KUKA KRL program: safety_test_01.src, safety_test_01.dat

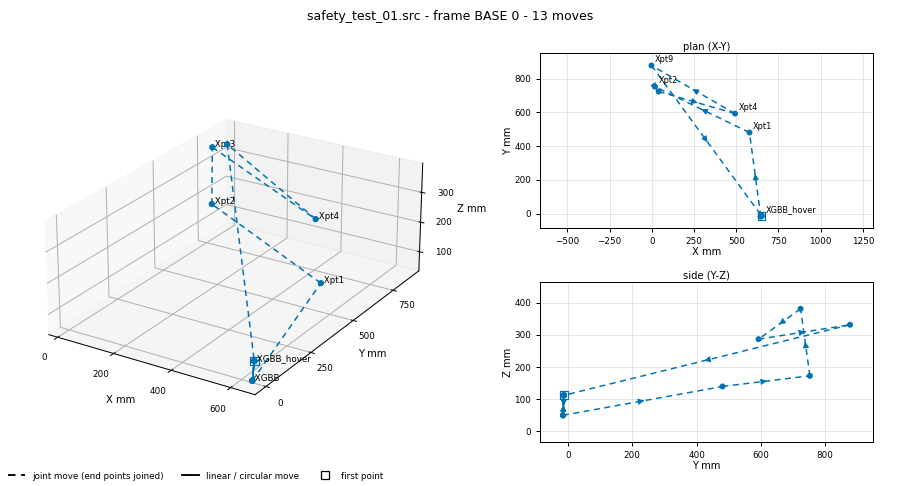
[picture p0: tool path of safety_test_01.src in frame BASE 0, 13 of 13 moves have a stored position in this frame; points joined in program order, loops and branches not executed]
--- safety_test_01.src ---
&ACCESS RVP
&REL 80
&PARAM TEMPLATE = C:\KRC\Roboter\Template\vorgabe
&PARAM EDITMASK = *
DEF safety_test_01( )

DECL INT COUNT
DECL INT MODE
DECL INT POSITION
DECL BOOL PREEMPT
DECL BOOL SICK_TEST
DECL BOOL STOP_TEST
DECL BOOL MOVING

;FOLD INI
  ;FOLD BASISTECH INI
    GLOBAL INTERRUPT DECL 3 WHEN $STOPMESS==TRUE DO IR_STOPM ( )
    INTERRUPT ON 3
    BAS (#INITMOV,0 )
  ;ENDFOLD (BASISTECH INI)
  ;FOLD USER INI
    ;Make your modifications here

  ;ENDFOLD (USER INI)
;ENDFOLD (INI)

; Start motions at the hover point
;FOLD PTP GBB_hover Vel=100 % PDAT1 Tool[4]:Pneumatic_gripper Base[0];%{PE}%R 5.6.11,%MKUKATPBASIS,%CMOVE,%VPTP,%P 1:PTP, 2:GBB_hover, 3:, 5:100, 7:PDAT1
$BWDSTART=FALSE
PDAT_ACT=PPDAT1
FDAT_ACT=FGBB_hover
BAS(#PTP_PARAMS,100)
PTP XGBB_hover
;ENDFOLD

MOVING=true
MODE = 4
POSITION = 1
PREEMPT = true
SICK_TEST = FALSE
STOP_TEST = FALSE

SWITCH MODE
  CASE 0
   ; SToP TeSt
   STOP_TEST = TRUE

  CASE 1
    ; Safety rated monitored stop
    OVERRIDE_SPEED = TRUE
    MOVE_PERMISSION = FALSE
  CASE 2
    ; Give permission for robot to move
    MOVE_PERMISSION = TRUE
    OVERRIDE_SPEED = FALSE
  CASE 3
    ; test 1
    MOVE_PERMISSION = FALSE
    OVERRIDE_SPEED = FALSe
  CASE 4
    ; full test
    OVERRIDE_SPEED = TRUE
    MOVE_PERMISSION = true
ENDSWITCH



; Move to button
;FOLD LIN GBB Vel=0.5 m/s CPDAT4 Tool[4]:Pneumatic_gripper Base[0];%{PE}%R 5.6.11,%MKUKATPBASIS,%CMOVE,%VLIN,%P 1:LIN, 2:GBB, 3:, 5:0.5, 7:CPDAT4
$BWDSTART=FALSE
LDAT_ACT=LCPDAT4
FDAT_ACT=FGBB
BAS(#CP_PARAMS,0.5)
LIN XGBB
;ENDFOLD

HALT

;FOLD WAIT Time=15 sec;%{PE}%R 5.6.11,%MKUKATPBASIS,%CWAIT,%VWAIT,%P 2:15
WAIT SEC 15
;ENDFOLD

; 2 stow request
; 3 robot can move
; 4 agv stopped
; 5 agv stopped verify
; 6 sick signal

IF SICK_TEST THEN
  WHILE TRUE
    IF $IN[6] THEN
      $OUT[1] = FALSE
    ELSE
      $OUT[1] = TRUE
    ENDIF
  ENDWHILE
ELSE
  IF MOVE_PERMISSION OR STOP_TEST THEN
;    $OUT[1] = TRUE
    IF MOVE_PERMISSION THEN
      ; Permission to move
      WAIT FOR ($IN[3])
    ENDIF
    ; Verification is safe to move
    WAIT FOR ($IN[4] and not $IN[5])

;    WAIT FOR ($IN[4])
  ENDIF

  ;FOLD PTP GBB_hover Vel=100 % PDAT15 Tool[4]:Pneumatic_gripper Base[0];%{PE}%R 5.6.11,%MKUKATPBASIS,%CMOVE,%VPTP,%P 1:PTP, 2:GBB_hover, 3:, 5:100, 7:PDAT15
$BWDSTART=FALSE
PDAT_ACT=PPDAT15
FDAT_ACT=FGBB_hover
BAS(#PTP_PARAMS,100)
PTP XGBB_hover
;ENDFOLD

;  HALT

  FOR COUNT = 1 TO 80
    ; Allow AGV to preempt motion
    IF (PREEMPT AND MOVE_PERMISSION) OR (STOP_TEST AND $IN[5]) THEN
      IF $IN[2] OR (STOP_TEST AND $IN[5]) THEN
;        PTP GBB_HOVER C_PTP

        ;FOLD PTP GBB_hover Vel=100 % PDAT16 Tool[4]:Pneumatic_gripper Base[0];%{PE}%R 5.6.11,%MKUKATPBASIS,%CMOVE,%VPTP,%P 1:PTP, 2:GBB_hover, 3:, 5:100, 7:PDAT16
$BWDSTART=FALSE
PDAT_ACT=PPDAT16
FDAT_ACT=FGBB_hover
BAS(#PTP_PARAMS,100)
PTP XGBB_hover
;ENDFOLD
;        LIN GBB

        ;FOLD LIN GBB Vel=0.5 m/s CPDAT5 Tool[4]:Pneumatic_gripper Base[0];%{PE}%R 5.6.11,%MKUKATPBASIS,%CMOVE,%VLIN,%P 1:LIN, 2:GBB, 3:, 5:0.5, 7:CPDAT5
$BWDSTART=FALSE
LDAT_ACT=LCPDAT5
FDAT_ACT=FGBB
BAS(#CP_PARAMS,0.5)
LIN XGBB
;ENDFOLD
        IF MOVE_PERMISSION THEN
          WAIT FOR ((NOT $IN[2]) and ($IN[3]))
        ELSE
          WAIT FOR ($IN[4] AND NOT $IN[5])
        ENDIF
      ENDIF
    ENDIF

    IF MOVING THEN
      SWITCH POSITION
      CASE 1
        ;FOLD PTP pt1 CONT Vel=50 % PDAT10 Tool[4]:Pneumatic_gripper Base[0];%{PE}%R 5.6.11,%MKUKATPBASIS,%CMOVE,%VPTP,%P 1:PTP, 2:pt1, 3:C_PTP, 5:50, 7:PDAT10
$BWDSTART=FALSE
PDAT_ACT=PPDAT10
FDAT_ACT=Fpt1
BAS(#PTP_PARAMS,50)
PTP Xpt1 C_PTP
;ENDFOLD
        POSITION = 2
      CASE 2
        ;FOLD PTP pt2 CONT Vel=50 % PDAT11 Tool[4]:Pneumatic_gripper Base[0];%{PE}%R 5.6.11,%MKUKATPBASIS,%CMOVE,%VPTP,%P 1:PTP, 2:pt2, 3:C_PTP, 5:50, 7:PDAT11
$BWDSTART=FALSE
PDAT_ACT=PPDAT11
FDAT_ACT=Fpt2
BAS(#PTP_PARAMS,50)
PTP Xpt2 C_PTP
;ENDFOLD
        POSITION = 3
      CASE 3
        ;FOLD PTP pt3 CONT Vel=50 % PDAT12 Tool[4]:Pneumatic_gripper Base[0];%{PE}%R 5.6.11,%MKUKATPBASIS,%CMOVE,%VPTP,%P 1:PTP, 2:pt3, 3:C_PTP, 5:50, 7:PDAT12
$BWDSTART=FALSE
PDAT_ACT=PPDAT12
FDAT_ACT=Fpt3
BAS(#PTP_PARAMS,50)
PTP Xpt3 C_PTP
;ENDFOLD
        POSITION = 4
      CASE 4
        ;FOLD PTP pt4 CONT Vel=50 % PDAT13 Tool[4]:Pneumatic_gripper Base[0];%{PE}%R 5.6.11,%MKUKATPBASIS,%CMOVE,%VPTP,%P 1:PTP, 2:pt4, 3:C_PTP, 5:50, 7:PDAT13
$BWDSTART=FALSE
PDAT_ACT=PPDAT13
FDAT_ACT=Fpt4
BAS(#PTP_PARAMS,50)
PTP Xpt4 C_PTP
;ENDFOLD
        POSITION = 1
      ENDSWITCH
    ELSE

;FOLD PTP pt9 Vel=50 % PDAT17 Tool[1]:flange_adapter Base[0];%{PE}%R 5.6.11,%MKUKATPBASIS,%CMOVE,%VPTP,%P 1:PTP, 2:pt9, 3:, 5:50, 7:PDAT17
$BWDSTART=FALSE
PDAT_ACT=PPDAT17
FDAT_ACT=Fpt9
BAS(#PTP_PARAMS,50)
PTP Xpt9
;ENDFOLD
    ENDIF
  ENDFOR


  $OUT[1] = FALSE
ENDIF

; move back to button
;FOLD PTP GBB_hover Vel=100 % PDAT9 Tool[4]:Pneumatic_gripper Base[0];%{PE}%R 5.6.11,%MKUKATPBASIS,%CMOVE,%VPTP,%P 1:PTP, 2:GBB_hover, 3:, 5:100, 7:PDAT9
$BWDSTART=FALSE
PDAT_ACT=PPDAT9
FDAT_ACT=FGBB_hover
BAS(#PTP_PARAMS,100)
PTP XGBB_hover
;ENDFOLD

;FOLD LIN GBB Vel=0.5 m/s CPDAT1 Tool[4]:Pneumatic_gripper Base[0];%{PE}%R 5.6.11,%MKUKATPBASIS,%CMOVE,%VLIN,%P 1:LIN, 2:GBB, 3:, 5:0.5, 7:CPDAT1
$BWDSTART=FALSE
LDAT_ACT=LCPDAT1
FDAT_ACT=FGBB
BAS(#CP_PARAMS,0.5)
LIN XGBB
;ENDFOLD

HALT

;FOLD PTP GBB_hover Vel=100 % PDAT2 Tool[4]:Pneumatic_gripper Base[0];%{PE}%R 5.6.11,%MKUKATPBASIS,%CMOVE,%VPTP,%P 1:PTP, 2:GBB_hover, 3:, 5:100, 7:PDAT2
$BWDSTART=FALSE
PDAT_ACT=PPDAT2
FDAT_ACT=FGBB_hover
BAS(#PTP_PARAMS,100)
PTP XGBB_hover
;ENDFOLD

END

--- safety_test_01.dat ---
&ACCESS RVP
&REL 80
&PARAM TEMPLATE = C:\KRC\Roboter\Template\vorgabe
&PARAM EDITMASK = *
DEFDAT  SAFETY_TEST_01
;FOLD EXTERNAL DECLARATIONS;%{PE}%MKUKATPBASIS,%CEXT,%VCOMMON,%P
;FOLD BASISTECH EXT;%{PE}%MKUKATPBASIS,%CEXT,%VEXT,%P
EXT  BAS (BAS_COMMAND  :IN,REAL  :IN )
DECL INT SUCCESS
;ENDFOLD (BASISTECH EXT)
;FOLD USER EXT;%{E}%MKUKATPUSER,%CEXT,%VEXT,%P
;Make here your modifications

;ENDFOLD (USER EXT)
;ENDFOLD (EXTERNAL DECLARATIONS)
DECL BASIS_SUGG_T LAST_BASIS={POINT1[] "pt9                     ",POINT2[] "pt9                     ",CP_PARAMS[] "CPDAT5                  ",PTP_PARAMS[] "PDAT17                  ",CONT[] "                        ",CP_VEL[] "0.5                     ",PTP_VEL[] "50                      ",SYNC_PARAMS[] "SYNCDAT                 ",SPL_NAME[] "S0                      "}
DECL E6POS XGBB={X 645.417786,Y -15.7424402,Z 49.9040794,A -176.547302,B -2.40271902,C -179.064407,S 6,T 57,E1 4.61637783,E2 0.0,E3 0.0,E4 0.0,E5 0.0,E6 0.0}
DECL FDAT FGBB={TOOL_NO 4,BASE_NO 0,IPO_FRAME #BASE,POINT2[] " ",TQ_STATE FALSE}
DECL LDAT LCPDAT1={VEL 2.0,ACC 100.0,APO_DIST 100.0,APO_FAC 50.0,ORI_TYP #VAR,CIRC_TYP #BASE,JERK_FAC 50.0,EXAX_IGN 0}
DECL E6POS XGBB_HOVER={X 649.790894,Y -12.6510601,Z 112.200302,A -176.0495,B -0.632367313,C 179.939606,S 6,T 57,E1 6.48830223,E2 0.0,E3 0.0,E4 0.0,E5 0.0,E6 0.0}
DECL FDAT FGBB_hover={TOOL_NO 4,BASE_NO 0,IPO_FRAME #BASE,POINT2[] " ",TQ_STATE FALSE}
DECL PDAT PPDAT1={VEL 100.0,ACC 100.0,APO_DIST 100.0,APO_MODE #CPTP}
DECL PDAT PPDAT2={VEL 100.0,ACC 100.0,APO_DIST 100.0,APO_MODE #CPTP}
DECL LDAT LCPDAT2={VEL 2.0,ACC 100.0,APO_DIST 100.0,APO_FAC 50.0,ORI_TYP #VAR,CIRC_TYP #BASE,JERK_FAC 50.0,EXAX_IGN 0}
DECL PDAT PPDAT3={VEL 100.0,ACC 100.0,APO_DIST 100.0,APO_MODE #CPTP}
DECL LDAT LCPDAT3={VEL 2.0,ACC 100.0,APO_DIST 100.0,APO_FAC 50.0,ORI_TYP #VAR,CIRC_TYP #BASE,JERK_FAC 50.0,EXAX_IGN 0}
DECL PDAT PPDAT4={VEL 100.0,ACC 100.0,APO_DIST 100.0,APO_MODE #CPTP}
DECL PDAT PPDAT5={VEL 100.0,ACC 100.0,APO_DIST 100.0,APO_MODE #CPTP}
DECL E6POS Xpt1={X 578.458191,Y 480.555115,Z 139.689499,A -115.749001,B 2.50130701,C 176.941299,S 6,T 56,E1 13.3937902,E2 0.0,E3 0.0,E4 0.0,E5 0.0,E6 0.0}
DECL FDAT Fpt1={TOOL_NO 4,BASE_NO 0,IPO_FRAME #BASE,POINT2[] " ",TQ_STATE FALSE}
DECL E6POS XPT2={X 18.7999401,Y 752.495117,Z 172.8591,A -81.8293762,B -0.0247380901,C -178.297607,S 6,T 56,E1 11.7572699,E2 0.0,E3 0.0,E4 0.0,E5 0.0,E6 0.0}
DECL FDAT Fpt2={TOOL_NO 4,BASE_NO 0,IPO_FRAME #BASE,POINT2[] " ",TQ_STATE FALSE}
DECL PDAT PPDAT6={VEL 100.0,ACC 100.0,APO_DIST 100.0,APO_MODE #CPTP}
DECL E6POS XPT3={X 40.6591415,Y 723.555603,Z 381.292511,A -85.5868073,B 2.55676007,C -177.368393,S 6,T 56,E1 11.7302399,E2 0.0,E3 0.0,E4 0.0,E5 0.0,E6 0.0}
DECL FDAT Fpt3={TOOL_NO 4,BASE_NO 0,IPO_FRAME #BASE,POINT2[] " ",TQ_STATE FALSE}
DECL PDAT PPDAT7={VEL 100.0,ACC 100.0,APO_DIST 100.0,APO_MODE #CPTP}
DECL E6POS XPT4={X 493.052887,Y 592.738525,Z 286.833893,A -98.5490112,B 2.87527895,C -176.283203,S 6,T 56,E1 11.7201405,E2 0.0,E3 0.0,E4 0.0,E5 0.0,E6 0.0}
DECL FDAT Fpt4={TOOL_NO 4,BASE_NO 0,IPO_FRAME #BASE,POINT2[] " ",TQ_STATE FALSE}
DECL PDAT PPDAT8={VEL 100.0,ACC 100.0,APO_DIST 100.0,APO_MODE #CPTP}
DECL PDAT PPDAT9={VEL 100.0,ACC 100.0,APO_DIST 100.0,APO_MODE #CPTP}
DECL PDAT PPDAT10={VEL 100.0,ACC 100.0,APO_DIST 100.0,APO_MODE #CPTP}
DECL E6POS Xpt5={X 649.790894,Y -12.6510601,Z 112.200302,A -176.0495,B -0.632367313,C 179.939606,S 6,T 57,E1 6.48830223,E2 0.0,E3 0.0,E4 0.0,E5 0.0,E6 0.0}
DECL FDAT Fpt5={TOOL_NO 4,BASE_NO 0,IPO_FRAME #BASE,POINT2[] " ",TQ_STATE FALSE}
DECL PDAT PPDAT11={VEL 100.0,ACC 100.0,APO_DIST 100.0,APO_MODE #CPTP}
DECL E6POS Xpt6={X 18.7999401,Y 752.495117,Z 172.8591,A -81.8293762,B -0.0247380901,C -178.297607,S 6,T 56,E1 11.7572699,E2 0.0,E3 0.0,E4 0.0,E5 0.0,E6 0.0}
DECL FDAT Fpt6={TOOL_NO 4,BASE_NO 0,IPO_FRAME #BASE,POINT2[] " ",TQ_STATE FALSE}
DECL PDAT PPDAT12={VEL 100.0,ACC 100.0,APO_DIST 100.0,APO_MODE #CPTP}
DECL E6POS Xpt7={X 40.6591415,Y 723.555603,Z 381.292511,A -85.5868073,B 2.55676007,C -177.368393,S 6,T 56,E1 11.7302399,E2 0.0,E3 0.0,E4 0.0,E5 0.0,E6 0.0}
DECL FDAT Fpt7={TOOL_NO 4,BASE_NO 0,IPO_FRAME #BASE,POINT2[] " ",TQ_STATE FALSE}
DECL PDAT PPDAT13={VEL 100.0,ACC 100.0,APO_DIST 100.0,APO_MODE #CPTP}
DECL E6POS Xpt8={X 493.052887,Y 592.738525,Z 286.833893,A -98.5490112,B 2.87527895,C -176.283203,S 6,T 56,E1 11.7201405,E2 0.0,E3 0.0,E4 0.0,E5 0.0,E6 0.0}
DECL FDAT Fpt8={TOOL_NO 4,BASE_NO 0,IPO_FRAME #BASE,POINT2[] " ",TQ_STATE FALSE}
DECL PDAT PPDAT14={VEL 100.0,ACC 100.0,APO_DIST 100.0,APO_MODE #CPTP}
DECL PDAT PPDAT15={VEL 100.0,ACC 100.0,APO_DIST 100.0,APO_MODE #CPTP}
DECL LDAT LCPDAT4={VEL 2.0,ACC 100.0,APO_DIST 100.0,APO_FAC 50.0,ORI_TYP #VAR,CIRC_TYP #BASE,JERK_FAC 50.0,EXAX_IGN 0}
DECL PDAT PPDAT16={VEL 100.0,ACC 100.0,APO_DIST 100.0,APO_MODE #CPTP}
DECL LDAT LCPDAT5={VEL 2.0,ACC 100.0,APO_DIST 100.0,APO_FAC 50.0,ORI_TYP #VAR,CIRC_TYP #BASE,JERK_FAC 50.0,EXAX_IGN 0}
DECL E6POS XPT9={X -1.69614697,Y 877.449829,Z 331.721893,A 37.6611595,B 85.6146164,C -52.4638901,S 2,T 40,E1 4.61754513,E2 0.0,E3 0.0,E4 0.0,E5 0.0,E6 0.0}
DECL FDAT Fpt9={TOOL_NO 1,BASE_NO 0,IPO_FRAME #BASE,POINT2[] " ",TQ_STATE FALSE}
DECL PDAT PPDAT17={VEL 100.0,ACC 100.0,APO_DIST 100.0,APO_MODE #CPTP}
ENDDAT
